// TIA Portal V20 export
DATA_BLOCK "LASERDIAG"   // DB45
{ S7_Optimized_Access := 'FALSE' }
VERSION : 0.1
// 표준 접근 : 그리퍼 레이저 센서 진단 (센서별 상태 / Z 오프셋 자동 교정 / 측정별 진단 이력). 갱신은 "UL_LaserDiag". gr-console 이 읽고 ZCal.Enable / Reset 을 쓴다, 레이아웃은 LayoutSig 로 검증
// stored: AutoNumber true, DBAccessibleFromOPCUA true, DBAccessibleFromWebserver true, IsOnlyStoredInLoadMemory false, IsWriteProtectedInAS false
   VAR
      LayoutSig : DWord := 16#2917_602B;   // 레이아웃 서명 (gr-contract gen-sig 가 생성, 수동 수정 금지)
      Reset : Bool;   // 센서 상태 / 진단 이력 초기화 (자동 해제). 센서 교체·재취부 후 사용
      Sensor { S7_SetPoint := 'True'} : Array[0..3] of "LGR_LaserSensorHealth";   // 방향별 상태 (0 L, 1 F, 2 R, 3 B)
      ZCal { S7_SetPoint := 'True'} : "LGR_LaserZCal";   // Z 오프셋 자동 교정 : ZCal.Enable 을 켜고 타이어 측정 반복
      Head : Int;   // 다음 기록 위치 (0..49 링버퍼, 최신 = Entry[Head-1])
      Count : Int;   // 유효 기록 수 (최대 50)
      Total : UDInt;   // 누적 기록 수 = 마지막 Seq
      Entry { S7_SetPoint := 'True'} : Array[0..49] of "LGR_LaserDiagEntry";   // 측정별 진단 이력
      Edge : Struct   // 측정 완료 에지 메모리
         PickDone : Bool;
         InDone : Bool;
         OutDone : Bool;
         ManualDone : Bool;
      END_STRUCT;
   END_VAR
BEGIN
END_DATA_BLOCK
